// TIA Portal V17 export
// export: Created 2022-07-20T07:01:28.2607985Z, ExportSetting WithDefaults, DisplayName Totally Integrated Automation Portal, DisplayVersion V17, DisplayName TIA Portal Openness, DisplayVersion V17, DisplayName TIA Portal Version Control Interface, DisplayVersion V17, DisplayName SINAMICS Startdrive Advanced, DisplayVersion V17, DisplayName SINAMICS Startdrive G130, G150, S120, S150, SINAMICS MV, S210, DisplayVersion V17, DisplayName SINAMICS Startdrive G110M, G120, G120C, G120D, G120P, G115D, DisplayVersion V17, DisplayName STEP 7 Professional, DisplayVersion V17, DisplayName STEP 7 Safety, DisplayVersion V17, DisplayName WinCC Advanced, DisplayVersion V17
FUNCTION_BLOCK "FB10182_ChuckPortionTracking"   // FB10182, LAD
{ S7_Optimized_Access := 'TRUE' }
VERSION : 0.1
// stored: AutoNumber false, IsIECCheckEnabled false, IsRetainMemResEnabled false, MemoryReserve 100, SetENOAutomatically false, UDAEnableTagReadback false
   VAR_INPUT
      EnablePortionTracking : Bool;
      StartPosition : Real;
      EndPosition : Real;
      ChuckActualPosition : Real;
   END_VAR
   VAR_OUTPUT
      StartPositionReached : Bool;
      EndPositionReached : Bool;
   END_VAR
   VAR
      PortionTravelCheckStateDiagram : Int;
      R_TRIG_EnableTracking : R_TRIG;
   END_VAR
   VAR CONSTANT
      "0_WAIT_FOR_CHUCK_PORTION_TRACKING" : Int := 0;
      "10_CHUCK_BEFORE_START_POSITION" : Int := 10;
      "20_CHUCK_AFTER_START_POSITION" : Int := 20;
      "30_CHUCK_AFTER_END_POSITION" : Int := 30;
      "40_CHUCK_PORTION_TRACKING_DONE" : Int := 40;
   END_VAR
BEGIN

REGION Network 1 (SCL): First Scan
   IF "FirstScan" THEN
       #StartPositionReached := FALSE;
       #EndPositionReached := FALSE;
       #PortionTravelCheckStateDiagram := #"0_WAIT_FOR_CHUCK_PORTION_TRACKING";
   END_IF;
END_REGION

REGION Network 2 (SCL): Edge Signals & Timers
   REGION EDGE SIGNALS
       #R_TRIG_EnableTracking(CLK := #EnablePortionTracking);
   END_REGION
END_REGION

REGION Network 3 (SCL): Tracking Management
   IF NOT (#EnablePortionTracking) THEN
       #StartPositionReached := FALSE;
       #EndPositionReached := FALSE;
       #PortionTravelCheckStateDiagram := #"0_WAIT_FOR_CHUCK_PORTION_TRACKING";
   END_IF;

   CASE #PortionTravelCheckStateDiagram OF
       #"0_WAIT_FOR_CHUCK_PORTION_TRACKING":
           IF #R_TRIG_EnableTracking.Q THEN
               #StartPositionReached := FALSE;
               #EndPositionReached := FALSE;
               #PortionTravelCheckStateDiagram := #"10_CHUCK_BEFORE_START_POSITION";
           END_IF;
       #"10_CHUCK_BEFORE_START_POSITION":
           IF #ChuckActualPosition < #StartPosition THEN
               #PortionTravelCheckStateDiagram := #"20_CHUCK_AFTER_START_POSITION";
           END_IF;
       #"20_CHUCK_AFTER_START_POSITION":
           IF #ChuckActualPosition > #StartPosition THEN
               #StartPositionReached := TRUE;
               #PortionTravelCheckStateDiagram := #"30_CHUCK_AFTER_END_POSITION";
           END_IF;
       #"30_CHUCK_AFTER_END_POSITION":
           IF #ChuckActualPosition > #EndPosition THEN
               #EndPositionReached := TRUE;
               #PortionTravelCheckStateDiagram := #"40_CHUCK_PORTION_TRACKING_DONE";
           END_IF;
       #"40_CHUCK_PORTION_TRACKING_DONE":
           #PortionTravelCheckStateDiagram := #"0_WAIT_FOR_CHUCK_PORTION_TRACKING";
   END_CASE;
END_REGION
END_FUNCTION_BLOCK
